{attribute 'GeneratedUsingTerminal: EL3681-0000-0017'}
{attribute addProperty BoxType "EL3681-0000-0017"}
{attribute addProperty Id "SAI_InputsAT %I*SAI_Inputs_3A838E1114SAI_RangeAT %I*SAI_Range_C3200E782SAI_Range_1AT %Q*SAI_Range_3710D7473WcStateAT %I*WcState_9091E0EB2InfoDataAT %I*InfoData_94A18F5E2"}
{attribute addProperty CRC "1207913307"}
{attribute addProperty Size "23"}
TYPE EL3681_47FF4B5B EXTENDS EtcSlaveTerminalBase_947E5A46 :
STRUCT
	{attribute addProperty Name "SAI_Inputs"}
	SAI_Inputs : SAI_Inputs_3A838E11;
	{attribute addProperty Name "SAI_Range"}
	SAI_Range : SAI_Range_C3200E78;
	{attribute addProperty Name "SAI_Range_1"}
	SAI_Range_1 : SAI_Range_3710D747;
	{attribute addProperty Name "WcState"}
	WcState : WcState_9091E0EB;
	{attribute addProperty Name "InfoData"}
	InfoData : InfoData_94A18F5E;
END_STRUCT
END_TYPE

(* stored: Version 1.2.0.0, ProductVersion 3.1.4024.9
   DUT EL3681_47FF4B5B: Id {99aee58e-393e-4623-95d1-0c074101c769} *)
